Fanuc KAREL source: UNPOS.kl

PROGRAM T
%NOLOCKGROUP
VAR
 v0 : XYZWPR
 v1 : REAL
 v2 : REAL
 v3 : REAL
 v4 : REAL
 v5 : REAL
 v6 : REAL
 v7 : CONFIG
BEGIN
 UNPOS(v0, v1, v2, v3, v4, v5, v6, v7)
END T
